// TIA Portal V20 export
FUNCTION "PositionAbsolute_No" : Void   // FC32780, LAD
// stored: Namespace Unit1.Em5, SetENOAutomatically false
BEGIN
END_FUNCTION
